% RSLogix 500 project SCP Analog Example.RSS, saved by version 8.30.00.16 %
PROJECT "UNTITLED"    % processor: Bul.1763 MicroLogix 1100 Series B %

PROGRAM FILES
  LAD 2   5 rungs

DATA FILES
  O0 OUTPUT  4 elements
  I1 INPUT  6 elements
  S2 STATUS  66 elements
  B3 BINARY  1 elements
  T4 TIMER  1 elements
  C5 COUNTER  1 elements
  R6 CONTROL  1 elements
  N7 INTEGER  4 elements
  F8 FLOAT  1 elements

LADDER 2
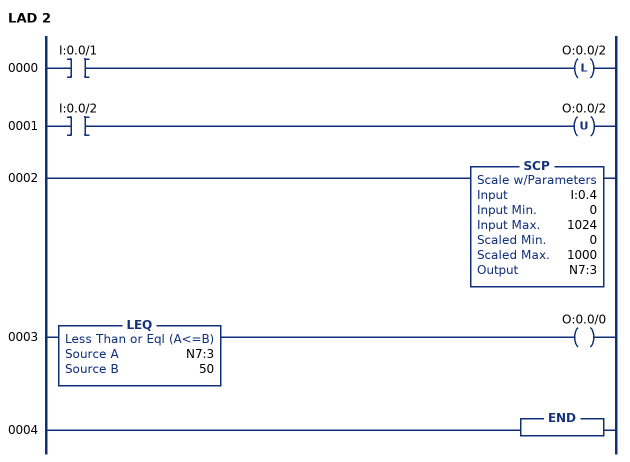
% Rung: 0 %
SOR XIC I:0.0/1 OTL O:0.0/2 EOR
% Rung: 1 %
SOR XIC I:0.0/2 OTU O:0.0/2 EOR
% Rung: 2 %
SOR SCP I:0.4 0 1024 0 1000 N7:3 EOR
% Rung: 3 %
SOR LEQ N7:3 50 OTE O:0.0/0 EOR
% Rung: 4 %
SOR END EOR

REVISION NOTES
  0: add counter

DATA TABLE (non-zero values as saved)
DATA T4
% .PRE .ACC %
% T4:0 % 5 0
DATA C5
% .PRE .ACC %
% C5:0 % 5 1
